Yaskawa INFORM job: OK_R2_O24B(90,0)KMOK.JBI

/JOB
//NAME OK_R2_O24B(90,0)KMOK
///FOLDERNAME X4
//POS
///NPOS 235,235,235,13,0,0
///TOOL 0
///POSTYPE PULSE
///PULSE
C00000=110421,-114568,-128442,17543,109310,-40994
C00001=110421,-114568,-128442,17543,109310,-40994
C00002=114535,-118016,-126260,17193,105500,-40103
C00003=116189,-118926,-125238,17079,104117,-39719
C00004=122470,-118801,-125267,16970,102934,-37675
C00005=122542,-119768,-123081,16831,101153,-37902
C00006=122470,-118801,-125267,16970,102934,-37675
C00007=116189,-118926,-125238,17079,104117,-39719
C00008=115768,-121709,-122546,16840,101244,-40278
C00009=119833,-121860,-122638,16796,100405,-38960
C00010=115768,-121709,-122546,16840,101244,-40278
C00011=116189,-118926,-125238,17079,104117,-39719
C00012=114535,-118016,-126260,17193,105500,-40103
C00013=110421,-114568,-128442,17543,109310,-40994
C00014=126378,-115954,-129597,-15290,109099,41008
C00015=122420,-119367,-127301,-14983,105339,40105
C00016=120830,-120251,-126232,-14883,103983,39719
C00017=114862,-120096,-125989,-14784,102865,37775
C00018=115075,-121077,-123808,-14669,101114,38064
C00019=114862,-120096,-125989,-14784,102865,37775
C00020=120830,-120251,-126232,-14883,103983,39719
C00021=121393,-120121,-122865,-14745,102140,40145
C00022=117360,-120220,-122765,-14697,101321,38836
C00023=121393,-120121,-122865,-14745,102140,40145
C00024=120830,-120251,-126232,-14883,103983,39719
C00025=122420,-119367,-127301,-14983,105339,40105
C00026=126378,-115954,-129597,-15290,109099,41008
C00027=68546,-106272,-120466,-15386,126682,61056
C00028=65872,-117617,-121364,-15125,121103,60799
C00029=65994,-124789,-121483,-14506,117628,61338
C00030=65994,-124776,-119887,-14364,116682,61464
C00031=64727,-121841,-121551,-15095,118908,60654
C00032=66354,-118147,-119193,-14717,119632,61205
C00033=63947,-125385,-121489,-15018,116968,60618
C00034=66354,-118147,-119193,-14717,119632,61205
C00035=67446,-114060,-119015,-14744,121753,61346
C00036=69995,-103128,-118158,-14981,127125,61604
C00037=43458,-109907,-123851,-22079,119459,51827
C00038=39582,-118676,-123782,-21672,114241,51374
C00039=37960,-121735,-123576,-21587,112243,51139
C00040=38039,-122241,-121246,-21299,110682,51473
C00041=37960,-121735,-123576,-21587,112243,51139
C00042=39439,-119560,-121458,-21353,112446,51673
C00043=35892,-124835,-123088,-21550,109947,50789
C00044=39439,-119560,-121458,-21353,112446,51673
C00045=41022,-116597,-121679,-21425,114395,51908
C00046=44803,-108153,-121807,-21787,119465,52368
C00047=46269,-104607,-116900,-14890,131588,81597
C00048=45575,-117487,-118566,-13929,126044,82146
C00049=45272,-122474,-119074,-13631,123805,82329
C00050=45097,-121786,-116375,-13476,122503,82429
C00051=45272,-122474,-119074,-13631,123805,82329
C00052=54794,-132635,-122270,-15461,117667,84057
C00053=51488,-139835,-124335,-16145,114686,83176
C00054=54794,-132635,-122270,-15461,117667,84057
C00055=54354,-108181,-111858,-18613,130239,82011
C00056=56948,-114588,-113873,-16794,128830,83498
C00057=54354,-108181,-111858,-18613,130239,82011
C00058=54354,-108181,-111858,-18613,105079,82011
C00059=125473,-127815,-125744,20402,114696,-66128
C00060=144354,-128645,-122856,20089,112993,-66444
C00061=144356,-128558,-121667,19978,112345,-66561
C00062=143692,-123642,-120175,20108,114021,-66516
C00063=144449,-128577,-122916,20120,113038,-66399
C00064=144368,-128510,-121483,19685,112887,-66475
C00065=144076,-129076,-121363,22700,108650,-60338
C00066=144065,-129172,-121967,22849,108765,-60054
C00067=145562,-127750,-121174,-10660,122518,-78224
C00068=145562,-127687,-120572,-10615,122186,-78189
C00069=144870,-122921,-119115,-11103,123620,-78631
C00070=145668,-127710,-121822,-10673,122944,-78224
C00071=145551,-127683,-120865,-10446,122273,-78190
C00072=145550,-127738,-121466,-10490,122609,-78224
C00073=145528,-127702,-122047,-10145,122795,-78223
C00074=145466,-127681,-122511,-8080,122804,-78067
C00075=145466,-127654,-121910,-8044,122451,-78039
C00076=144776,-122735,-120395,-8485,123961,-78447
C00077=145489,-127675,-123160,-8112,123205,-78089
C00078=145462,-127615,-121976,-8108,122518,-78051
C00079=145461,-127639,-122576,-8144,122872,-78079
C00080=145470,-127509,-122616,-9202,123100,-78187
C00081=145470,-127489,-122014,-9161,122745,-78155
C00082=144781,-122556,-120500,-9628,124248,-78581
C00083=145526,-127464,-123250,-9229,123515,-78201
C00084=145457,-127452,-122138,-8905,122802,-78142
C00085=145457,-127468,-122738,-8946,123159,-78173
C00086=145419,-127422,-123013,-7792,123191,-78085
C00087=145369,-127281,-122655,-6352,123642,-78005
C00088=145369,-127269,-122086,-6324,123301,-77983
C00089=144684,-122332,-120516,-6740,124807,-78367
C00090=145346,-127303,-123341,-6395,124049,-78040
C00091=145359,-127218,-122002,-6175,123337,-77977
C00092=145359,-127231,-122569,-6203,123677,-77998
C00093=145369,-127141,-122578,-7278,123283,-78064
C00094=145369,-127129,-121996,-7245,122933,-78039
C00095=144683,-122199,-120454,-7674,124442,-78435
C00096=145369,-127140,-123243,-7317,123689,-78093
C00097=145374,-127101,-121995,-7642,122781,-78062
C00098=145373,-127113,-122583,-7677,123134,-78088
C00099=145323,-127035,-122273,-5816,123755,-77984
C00100=145301,-126904,-121478,-4974,124764,-77984
C00101=145245,-126972,-122476,-3510,122733,-77759
C00102=145245,-126962,-121900,-3495,122385,-77747
C00103=144566,-122041,-120337,-3835,123918,-78081
C00104=145130,-127078,-123177,-3572,123105,-77819
C00105=145235,-126936,-121864,-3341,122099,-77723
C00106=145235,-126947,-122445,-3356,122451,-77734
C00107=145235,-126704,-121159,-4007,122972,-77833
C00108=145235,-126667,-120590,-3990,122642,-77820
C00109=144560,-121896,-119039,-4346,124100,-78159
C00110=145144,-126819,-121880,-4063,123351,-77885
C00111=145222,-126734,-121009,-3552,122070,-77754
C00112=143543,-128240,-121764,-3717,120897,-78337
C00113=144110,-127812,-122791,-3542,121772,-78139
C00114=145205,-126597,-125313,-3216,123991,-77765
C00115=78497,-119087,-126940,8466,133839,-13526
C00116=78488,-120793,-123596,8031,130934,-13800
C00117=78485,-121192,-122172,7887,129863,-13894
C00118=78455,-120845,-123307,7986,130735,-13833
C00119=77443,-125885,-123641,7190,128464,-14473
C00120=78479,-121212,-122221,7886,129884,-13896
C00121=78482,-120810,-123644,8031,130956,-13801
C00122=78491,-119095,-126985,8467,133863,-13526
C00123=78416,-117369,-129459,-12992,98157,-11559
C00124=78415,-119818,-126610,-12888,95218,-11250
C00125=78415,-120492,-125378,-12858,94139,-11138
C00126=77369,-125600,-126977,-12690,92378,-11308
C00127=78323,-119762,-126393,-12873,95102,-11269
C00128=78420,-120510,-125276,-12857,94070,-11129
C00129=78420,-119847,-126511,-12886,95145,-11241
C00130=78422,-117430,-129370,-12989,98073,-11548
C00131=84214,-85469,-118328,-4842,91147,-7442
C00132=74059,-12147,-76922,-1404,102997,-10572
C00133=133925,-71820,-61688,34619,64887,-29675
C00134=146663,-27707,-36323,28508,66625,-23960
C00135=151246,10085,-12654,25869,69264,-21358
C00136=159319,6651,-31532,14872,93153,-16403
C00137=161049,12617,-24359,-3467,88226,-17180
C00138=159447,19004,-16554,-3012,86648,-17647
C00139=159447,18503,-15222,-3010,85575,-17623
C00140=159447,19004,-16554,-3012,86648,-17647
C00141=159431,21694,-14016,-3008,86468,-17647
C00142=159447,19004,-16554,-3012,86648,-17647
C00143=160658,9490,-26043,14512,91068,-16216
C00144=162575,15072,-19202,14033,89453,-15776
C00145=163627,18223,-16292,13777,89114,-15470
C00146=163448,17947,-16551,13818,89157,-15522
C00147=163448,17469,-15177,13812,88099,-15642
C00148=162575,15072,-19202,14033,89453,-15776
C00149=162575,15072,-19202,14033,89453,-15776
C00150=161695,11045,-24734,14261,90891,-15899
C00151=160389,8166,-30281,14612,92983,-16078
C00152=166173,5650,-32242,20871,98882,-24992
C00153=168031,7092,-27994,20429,96691,-24741
C00154=171973,10796,-22826,19648,94585,-23756
C00155=171973,10387,-21674,19614,93717,-23897
C00156=171973,10796,-22826,19648,94585,-23756
C00157=173021,12834,-20995,19450,94274,-23449
C00158=171973,10796,-22826,19648,94585,-23756
C00159=169411,6672,-28771,20198,96619,-24285
C00160=169457,3960,-30994,23440,104028,-32838
C00161=170821,3186,-27404,27142,100799,-32384
C00162=170821,2940,-26605,27078,100248,-32515
C00163=170821,3186,-27404,27142,100799,-32384
C00164=171855,3656,-27002,27037,100474,-32081
C00165=170821,3186,-27404,27142,100799,-32384
C00166=171453,4765,-27678,27184,101480,-31989
C00167=155920,16768,-644,63423,123153,25810
C00168=153914,19171,3953,62063,123660,24610
C00169=157147,16214,3501,61820,121007,24650
C00170=157145,16372,4776,61403,120658,24311
C00171=157147,16214,3501,61820,121007,24650
C00172=158673,15787,3108,62073,120051,24962
C00173=157147,16214,3501,61820,121007,24650
C00174=154267,18481,3545,62056,123385,24630
C00175=160586,-4724,-32336,44114,114513,18408
C00176=159707,-1654,-23897,45976,117158,-10277
C00177=160426,-1772,-22346,45643,116076,-10462
C00178=160426,-1854,-21195,45350,115539,-10739
C00179=160426,-1772,-22346,45643,116076,-10462
C00180=161004,-2697,-23104,45705,115781,-10311
C00181=160426,-1772,-22346,45643,116076,-10462
C00182=174615,37008,-2722,25510,99744,-54261
C00183=172498,42405,8067,32730,102732,-53174
C00184=172498,42136,9154,32614,102046,-53379
C00185=172498,42405,8067,32730,102732,-53174
C00186=173166,39976,5518,32734,102755,-52903
C00187=172498,42405,8067,32730,102732,-53174
C00188=171464,48985,12939,32850,103438,-53371
C00189=169687,51444,12946,33160,105162,-53551
C00190=164203,-2216,-38598,32315,111910,-16095
C00191=166391,-1836,-35337,31828,109592,-15933
C00192=166612,13037,-20307,31307,106989,-15305
C00193=163905,10722,-24642,31867,110359,-16693
C00194=163023,10318,-23737,31712,110017,-17150
C00195=166579,13090,-20261,31308,106999,-15315
C00196=166501,27487,-9192,25512,104586,-16954
C00197=162952,34148,-2586,21763,97726,-15315
C00198=160142,17407,-18468,27124,95473,-4322
C00199=163018,-2778,-39064,26713,96671,-3025
C00200=164611,45054,6259,27542,116257,-62631
C00201=165962,40795,4672,27363,114755,-62481
C00202=169650,39468,5367,27407,112609,-61559
C00203=167727,42077,8101,27182,112908,-62250
C00204=168804,38233,1799,27701,114270,-61464
C00205=172646,46850,13078,27417,110817,-60826
C00206=175258,53962,20871,27351,108970,-60262
C00207=175286,54040,20958,27350,108949,-60256
C00208=176029,42421,9462,27228,100378,-50913
C00209=177057,44715,12834,27836,95407,-46661
C00210=174286,53569,18433,27340,100959,-51234
C00211=172614,55478,17651,27620,102791,-51416
C00212=158797,4213,-33188,27539,97918,-4223
C00213=160288,6924,-27895,27122,95799,-4194
C00214=161417,15198,-18304,26815,93980,-4213
C00215=160867,8461,-26639,27014,95638,-4024
C00216=160120,6892,-26748,27110,95204,-4392
C00217=161403,15259,-18249,26817,93982,-4218
C00218=160305,12086,-21204,20161,86451,4179
C00219=159689,11147,-21822,11042,81082,13112
C00220=158372,16674,-18680,7008,84648,12184
C00221=156002,16176,-19181,4250,84243,10833
C00222=159539,6079,-28636,11078,82663,13207
C00223=159574,4391,-38688,11011,87883,13681
C00224=158609,-20032,-50850,30856,115372,-43029
C00225=166404,-23641,-48444,30293,109810,-41499
C00226=167846,-166,-34046,28078,125353,-30479
C00227=167052,574,-32162,27620,124908,-30970
C00228=166419,-23641,-48461,30296,109814,-41492
C00229=164454,-27920,-49253,33885,103588,-43249
C00230=166369,-22686,-46969,33128,99976,-43386
C00231=169987,-10838,-39904,28688,98031,-37107
C00232=168025,-24410,-44140,30807,78602,-40011
C00233=160117,-23281,-55166,26476,98061,-35003
C00234=156670,-29522,-57811,32418,104336,-21012
BC00000=365719,492449,1075139
BC00001=365719,363190,1075139
BC00002=365719,363190,1075139
BC00003=365719,363190,1075139
BC00004=365719,363190,1075139
BC00005=365719,363190,1075139
BC00006=365719,363190,1075139
BC00007=365719,363190,1075139
BC00008=365719,363190,1075139
BC00009=365719,363190,1075139
BC00010=365719,363190,1075139
BC00011=365719,363190,1075139
BC00012=365719,363190,1075139
BC00013=365719,363190,1075139
BC00014=303651,361671,1075139
BC00015=303651,361671,1075139
BC00016=303651,361671,1075139
BC00017=303651,361671,1075139
BC00018=303651,361671,1075139
BC00019=303651,361671,1075139
BC00020=303651,361671,1075139
BC00021=303651,361671,1075139
BC00022=303651,361671,1075139
BC00023=303651,361671,1075139
BC00024=303651,361671,1075139
BC00025=303651,361671,1075139
BC00026=303651,361671,1075139
BC00027=337725,299685,1075139
BC00028=337725,299685,1075139
BC00029=337725,299685,1075139
BC00030=337725,299685,1075139
BC00031=337725,299685,1075139
BC00032=337725,299685,1075139
BC00033=337725,299685,1075139
BC00034=337725,299685,1075139
BC00035=337725,299685,1075139
BC00036=337725,299685,1075139
BC00037=224410,277346,1075139
BC00038=224410,277346,1075139
BC00039=224410,277346,1075139
BC00040=224410,277346,1075139
BC00041=224410,277346,1075139
BC00042=224410,277346,1075139
BC00043=224410,277346,1075139
BC00044=224410,277346,1075139
BC00045=224410,277346,1075139
BC00046=224410,277346,1075139
BC00047=171285,286904,1075139
BC00048=171285,286904,1075139
BC00049=171285,286904,1075139
BC00050=171285,286904,1075139
BC00051=171285,286904,1075139
BC00052=171285,286904,1075139
BC00053=171285,286904,1075139
BC00054=171285,286904,1075139
BC00055=171285,286904,1075139
BC00056=171285,286904,1075139
BC00057=171285,286904,1075139
BC00058=171285,286904,1075139
BC00059=269590,309617,1075139
BC00060=267805,314819,1075139
BC00061=267092,316899,1075139
BC00062=267092,316899,1075139
BC00063=267092,316899,1075139
BC00064=264540,316051,1075139
BC00065=269908,321406,1075139
BC00066=270630,320628,1075139
BC00067=229341,315661,1075139
BC00068=229396,316752,1075139
BC00069=229396,316752,1075139
BC00070=229396,316752,1075139
BC00071=236075,316791,1075139
BC00072=236027,315702,1075139
BC00073=249293,315797,1075139
BC00074=258915,315256,1075139
BC00075=258916,316331,1075139
BC00076=258916,316331,1075139
BC00077=258916,316331,1075139
BC00078=265201,316325,1075139
BC00079=265198,315250,1075139
BC00080=282635,315456,1075139
BC00081=282673,316525,1075139
BC00082=282673,316525,1075139
BC00083=282673,316525,1075139
BC00084=289448,316439,1075139
BC00085=289419,315369,1075139
BC00086=298136,315044,1075139
BC00087=312054,313301,1075139
BC00088=312047,314425,1075139
BC00089=312047,314425,1075139
BC00090=312047,314425,1075139
BC00091=318602,314234,1075139
BC00092=318613,313105,1075139
BC00093=336310,314307,1075139
BC00094=336328,315407,1075139
BC00095=336328,315407,1075139
BC00096=336328,315407,1075139
BC00097=342205,315848,1075139
BC00098=342175,314758,1075139
BC00099=344940,312597,1075139
BC00100=345730,309912,1075139
BC00101=367542,313335,1075139
BC00102=367491,314445,1075139
BC00103=367491,314445,1075139
BC00104=367491,314445,1075139
BC00105=374233,314799,1075139
BC00106=374293,313698,1075139
BC00107=391653,312000,1075139
BC00108=391630,313137,1075139
BC00109=391630,313137,1075139
BC00110=391630,313137,1075139
BC00111=394304,314202,1075139
BC00112=398158,315264,1075139
BC00113=398158,313163,1075139
BC00114=397780,307912,1075139
BC00115=322189,319410,1075139
BC00116=319334,319411,1075139
BC00117=318192,319412,1075139
BC00118=318192,319412,1075139
BC00119=318192,319412,1075139
BC00120=313651,319426,1075139
BC00121=314793,319425,1075139
BC00122=317648,319424,1075139
BC00123=260501,369489,1075139
BC00124=262854,366425,1075139
BC00125=263796,365199,1075139
BC00126=263796,365199,1075139
BC00127=263796,365199,1075139
BC00128=267671,365187,1075139
BC00129=266729,366413,1075139
BC00130=264376,369477,1075139
BC00131=264376,420432,1075139
BC00132=221796,515972,1075139
BC00133=202683,509615,271551
BC00134=202683,475987,185561
BC00135=202683,457833,139139
BC00136=138971,364074,115966
BC00137=138971,364074,115966
BC00138=138971,364074,115966
BC00139=138971,364074,115966
BC00140=138971,364074,115966
BC00141=138971,364074,115966
BC00142=138971,364074,115966
BC00143=138971,364074,115966
BC00144=138971,364074,115966
BC00145=138971,364074,115966
BC00146=138971,364074,115966
BC00147=138971,364074,115966
BC00148=138971,364074,115966
BC00149=138971,364074,115966
BC00150=138971,364074,115966
BC00151=138971,364074,115966
BC00152=150418,367609,116980
BC00153=150418,367609,116980
BC00154=150418,367608,116974
BC00155=150418,367608,116974
BC00156=150418,367608,116974
BC00157=150418,367608,116974
BC00158=150418,367608,116974
BC00159=150418,367609,116980
BC00160=147886,366442,115691
BC00161=147886,366442,115691
BC00162=147886,366442,115691
BC00163=147886,366442,115691
BC00164=147886,366442,115691
BC00165=147886,366442,115691
BC00166=163814,366442,115691
BC00167=140803,365672,114840
BC00168=140803,365672,114840
BC00169=140803,365673,114838
BC00170=140803,365673,114838
BC00171=140803,365673,114838
BC00172=140803,365673,114838
BC00173=140803,365673,114838
BC00174=140803,365672,114840
BC00175=149676,372426,112080
BC00176=161597,381499,108373
BC00177=161597,381499,108373
BC00178=161597,381499,108373
BC00179=161597,381499,108373
BC00180=161597,381499,108373
BC00181=161597,381499,108373
BC00182=245846,421854,91883
BC00183=245846,421854,91881
BC00184=245846,421854,91881
BC00185=245846,421854,91881
BC00186=245846,421854,91881
BC00187=245846,421854,91881
BC00188=245846,421854,91883
BC00189=245846,421854,91883
BC00190=140778,359593,95378
BC00191=140778,359593,95378
BC00192=140779,374954,95371
BC00193=140778,374954,95378
BC00194=140778,374954,95378
BC00195=140779,374954,95371
BC00196=140779,374954,95375
BC00197=140779,374954,95372
BC00198=140778,374954,95378
BC00199=140778,365135,95378
BC00200=224235,422354,101557
BC00201=224235,422354,101557
BC00202=224235,422354,101557
BC00203=224235,422354,101557
BC00204=224235,422354,101557
BC00205=224235,422354,101557
BC00206=224235,422354,101557
BC00207=224235,422354,101557
BC00208=224235,422354,101557
BC00209=224235,422354,101557
BC00210=224235,422354,101557
BC00211=224235,422354,101557
BC00212=135486,365173,95416
BC00213=135486,365173,95416
BC00214=135486,365173,95416
BC00215=135486,365173,95416
BC00216=135486,365173,95416
BC00217=135486,365173,95416
BC00218=135486,365173,95416
BC00219=135487,365173,95415
BC00220=135487,365173,95415
BC00221=135487,365173,95415
BC00222=135486,365173,95416
BC00223=135486,365173,95416
BC00224=147706,371102,95331
BC00225=147706,371102,95331
BC00226=147707,371103,95336
BC00227=147707,371103,95336
BC00228=147706,371102,95331
BC00229=147706,371102,95331
BC00230=147706,371102,95331
BC00231=147706,371102,95331
BC00232=147706,371102,95331
BC00233=147706,371102,95331
BC00234=147707,371103,95336
EC00000=-798156,-183832
EC00001=-798156,-183832
EC00002=-798156,-183832
EC00003=-798156,-183832
EC00004=-798156,-183832
EC00005=-798156,-183832
EC00006=-798156,-183832
EC00007=-798156,-183832
EC00008=-798156,-183832
EC00009=-798156,-183832
EC00010=-798156,-183832
EC00011=-798156,-183832
EC00012=-798156,-183832
EC00013=-798156,-183832
EC00014=-798156,-183832
EC00015=-798156,-183832
EC00016=-798156,-183832
EC00017=-798156,-183832
EC00018=-798156,-183832
EC00019=-798156,-183832
EC00020=-798156,-183832
EC00021=-798156,-183832
EC00022=-798156,-183832
EC00023=-798156,-183832
EC00024=-798156,-183832
EC00025=-798156,-183832
EC00026=-798156,-183832
EC00027=-798156,-183832
EC00028=-798156,-183832
EC00029=-798156,-183832
EC00030=-798156,-183832
EC00031=-798156,-183832
EC00032=-798156,-183832
EC00033=-798156,-183832
EC00034=-798156,-183832
EC00035=-798156,-183832
EC00036=-798156,-183832
EC00037=-798156,-183832
EC00038=-798156,-183832
EC00039=-798156,-183832
EC00040=-798156,-183832
EC00041=-798156,-183832
EC00042=-798156,-183832
EC00043=-798156,-183832
EC00044=-798156,-183832
EC00045=-798156,-183832
EC00046=-798156,-183832
EC00047=-798156,-183832
EC00048=-798156,-183832
EC00049=-798156,-183832
EC00050=-798156,-183832
EC00051=-798156,-183832
EC00052=-798156,-183832
EC00053=-798156,-183832
EC00054=-798156,-183832
EC00055=-798156,-183832
EC00056=-798156,-183832
EC00057=-798156,-183832
EC00058=-798156,-183832
EC00059=-798156,-183832
EC00060=-798156,-183832
EC00061=-798156,-183832
EC00062=-798156,-183832
EC00063=-798156,-183832
EC00064=-798156,-183832
EC00065=-798156,-183832
EC00066=-798156,-183832
EC00067=-798156,-183832
EC00068=-798156,-183832
EC00069=-798156,-183832
EC00070=-798156,-183832
EC00071=-798156,-183832
EC00072=-798156,-183832
EC00073=-798156,-183832
EC00074=-798156,-183832
EC00075=-798156,-183832
EC00076=-798156,-183832
EC00077=-798156,-183832
EC00078=-798156,-183832
EC00079=-798156,-183832
EC00080=-798156,-183832
EC00081=-798156,-183832
EC00082=-798156,-183832
EC00083=-798156,-183832
EC00084=-798156,-183832
EC00085=-798156,-183832
EC00086=-798156,-183832
EC00087=-798156,-183832
EC00088=-798156,-183832
EC00089=-798156,-183832
EC00090=-798156,-183832
EC00091=-798156,-183832
EC00092=-798156,-183832
EC00093=-798156,-183832
EC00094=-798156,-183832
EC00095=-798156,-183832
EC00096=-798156,-183832
EC00097=-798156,-183832
EC00098=-798156,-183832
EC00099=-798156,-183832
EC00100=-798156,-183832
EC00101=-798156,-183832
EC00102=-798156,-183832
EC00103=-798156,-183832
EC00104=-798156,-183832
EC00105=-798156,-183832
EC00106=-798156,-183832
EC00107=-798156,-183832
EC00108=-798156,-183832
EC00109=-798156,-183832
EC00110=-798156,-183832
EC00111=-798156,-183832
EC00112=-798156,-183832
EC00113=-798156,-183832
EC00114=-798156,-183832
EC00115=-798156,-183832
EC00116=-798156,-183832
EC00117=-798156,-183832
EC00118=-798156,-183832
EC00119=-798156,-183832
EC00120=-798156,-183832
EC00121=-798156,-183832
EC00122=-798156,-183832
EC00123=-798156,-183832
EC00124=-798156,-183832
EC00125=-798156,-183832
EC00126=-798156,-183832
EC00127=-798156,-183832
EC00128=-798156,-183832
EC00129=-798156,-183832
EC00130=-798156,-183832
EC00131=-798156,-183832
EC00132=-798156,-183832
EC00133=-798156,-183832
EC00134=-798156,-183832
EC00135=-798156,-183832
EC00136=-798156,-183832
EC00137=-798156,-183832
EC00138=-798156,-183832
EC00139=-798156,-183832
EC00140=-798156,-183832
EC00141=-798156,-183832
EC00142=-798156,-183832
EC00143=-798156,-183832
EC00144=-798156,-183832
EC00145=-798156,-183832
EC00146=-798156,-183832
EC00147=-798156,-183832
EC00148=-798156,-183832
EC00149=-798156,-183832
EC00150=-798156,-183832
EC00151=-798156,-183832
EC00152=-798156,-183832
EC00153=-798156,-183832
EC00154=-798154,-183833
EC00155=-798154,-183833
EC00156=-798154,-183833
EC00157=-798154,-183833
EC00158=-798154,-183833
EC00159=-798156,-183832
EC00160=-798156,-183832
EC00161=-798156,-183832
EC00162=-798156,-183832
EC00163=-798156,-183832
EC00164=-798156,-183832
EC00165=-798156,-183832
EC00166=-798156,-183832
EC00167=-798156,-183832
EC00168=-798156,-183832
EC00169=-798154,-183832
EC00170=-798154,-183832
EC00171=-798154,-183832
EC00172=-798154,-183832
EC00173=-798154,-183832
EC00174=-798156,-183832
EC00175=-798156,-183832
EC00176=-798156,-183832
EC00177=-798156,-183832
EC00178=-798156,-183832
EC00179=-798156,-183832
EC00180=-798156,-183832
EC00181=-798156,-183832
EC00182=-798156,-183832
EC00183=-798154,-183833
EC00184=-798154,-183833
EC00185=-798154,-183833
EC00186=-798154,-183833
EC00187=-798154,-183833
EC00188=-798156,-183832
EC00189=-798156,-183832
EC00190=-798156,-183832
EC00191=-798156,-183832
EC00192=-798154,-183833
EC00193=-798156,-183832
EC00194=-798156,-183832
EC00195=-798154,-183833
EC00196=-798155,-183833
EC00197=-798154,-183834
EC00198=-798156,-183832
EC00199=-798156,-183832
EC00200=-798156,-183832
EC00201=-798156,-183832
EC00202=-798156,-183832
EC00203=-798156,-183832
EC00204=-798156,-183832
EC00205=-798156,-183832
EC00206=-798156,-183832
EC00207=-798156,-183832
EC00208=-798156,-183832
EC00209=-798156,-183832
EC00210=-798156,-183832
EC00211=-798156,-183832
EC00212=-798156,-183832
EC00213=-798156,-183832
EC00214=-798156,-183832
EC00215=-798156,-183832
EC00216=-798156,-183832
EC00217=-798156,-183832
EC00218=-798156,-183832
EC00219=-798155,-183833
EC00220=-798155,-183833
EC00221=-798155,-183833
EC00222=-798156,-183832
EC00223=-798156,-183832
EC00224=-798153,-183833
EC00225=-798153,-183833
EC00226=-798156,-183832
EC00227=-798156,-183832
EC00228=-798153,-183833
EC00229=-798153,-183833
EC00230=-798153,-183833
EC00231=-798153,-183833
EC00232=-798153,-183833
EC00233=-798153,-183833
EC00234=-798156,-183832
///POSTYPE BASE
///RECTAN
///RCONF 0,0,0,0,1,0,0,0,0,0,0,0,0,0,0,0,0,0,0,0,0,0,0,0
P00006=2.006,1.622,-0.565,0.0000,0.0000,0.0000
P00021=0.073,2.058,-0.109,0.0000,0.0000,0.0000
P00022=2.006,1.622,-0.565,0.0000,0.0000,0.0000
///RCONF 0,0,0,0,0,0,0,0,0,0,0,0,0,0,0,0,0,0,0,0,0,0,0,0
P00023=-2.957,-4.083,2.762,0.0000,0.0000,0.0000
P00024=-1.466,-0.226,-0.419,0.0000,0.0000,0.0000
P00025=3.643,0.007,-2.585,0.0000,0.0000,0.0000
P00026=2.644,0.055,-2.583,0.0000,0.0000,0.0000
P00027=2.278,0.099,-4.210,0.0000,0.0000,0.0000
P00031=-0.170,0.039,-0.647,0.0000,0.0000,0.0000
P00032=-0.423,0.157,3.222,0.0000,0.0000,0.0000
P00033=0.854,-1.099,3.047,0.0000,0.0000,0.0000
///RCONF 0,0,0,0,1,0,0,0,0,0,0,0,0,0,0,0,0,0,0,0,0,0,0,0
P00034=-8.151,9.743,-4.393,0.0000,0.0000,0.0000
///RCONF 0,0,0,0,0,0,0,0,0,0,0,0,0,0,0,0,0,0,0,0,0,0,0,0
P00035=0.390,-0.027,1.040,0.0000,0.0000,0.0000
//INST
///DATE 2024/11/18 12:50
///ATTR SC,RW
///GROUP1 RB1,BS1
///GROUP2 ST1
NOP
'OK_r2_O24B(90,0)
'
'brak tej czesci na razie
'Path S3723
SFTOF3D
MOVJ C00000 BC00000 VJ=100.00  +MOVJ EC00000 VJ=100.00
JUMP *LABEL
MOVJ C00001 BC00001 VJ=100.00  +MOVJ EC00001 VJ=100.00
MOVL C00002 BC00002 V=400.0  +MOVJ EC00002 VJ=100.00
SMOVL C00003 BC00003 V=100.0  +MOVJ EC00003
'BRAK DETALU
PAUSE
SMOVL C00004 BC00004 V=60.0  +MOVJ EC00004
SREFP 3 C00005 BC00005  +REFP EC00005
CALL JOB:SEARCH-R1-S13D
SET P031 P006
SFTON3D P031
SMOVL C00006 BC00006 V=60.0  +MOVJ EC00006
SMOVL C00007 BC00007 V=100.0  +MOVJ EC00007
SMOVL C00008 BC00008 V=60.0  +MOVJ EC00008
SREFP 3 C00009 BC00009  +REFP EC00009
CALL JOB:SEARCH-R1-S13D
SET P031 P006
SFTON3D P031
SMOVL C00010 BC00010 V=60.0  +MOVJ EC00010
SMOVL C00011 BC00011 V=100.0  +MOVJ EC00011
MOVL C00012 BC00012 V=400.0  +MOVJ EC00012 VJ=100.00
MOVL C00013 BC00013 V=1000.0  +MOVJ EC00013 VJ=100.00
'Path S3724
SFTOF3D
MOVJ C00014 BC00014 VJ=100.00  +MOVJ EC00014 VJ=100.00
MOVL C00015 BC00015 V=400.0  +MOVJ EC00015 VJ=100.00
SMOVL C00016 BC00016 V=100.0  +MOVJ EC00016
SMOVL C00017 BC00017 V=60.0  +MOVJ EC00017
SREFP 3 C00018 BC00018  +REFP EC00018
CALL JOB:SEARCH-R1-S13D
SET P032 P006
SFTON3D P032
SMOVL C00019 BC00019 V=60.0  +MOVJ EC00019
SMOVL C00020 BC00020 V=100.0  +MOVJ EC00020
SMOVL C00021 BC00021 V=60.0  +MOVJ EC00021
SREFP 3 C00022 BC00022  +REFP EC00022
CALL JOB:SEARCH-R1-S13D
SET P032 P006
SFTON3D P032
SMOVL C00023 BC00023 V=60.0  +MOVJ EC00023
SMOVL C00024 BC00024 V=100.0  +MOVJ EC00024
MOVL C00025 BC00025 V=400.0  +MOVJ EC00025 VJ=100.00
MOVL C00026 BC00026 V=1000.0  +MOVJ EC00026 VJ=100.00
'Path S3725
SFTOF3D
MOVJ C00027 BC00027 VJ=100.00  +MOVJ EC00027 VJ=100.00
MOVL C00028 BC00028 V=400.0  +MOVJ EC00028 VJ=100.00
SMOVL C00029 BC00029 V=60.0  +MOVJ EC00029
SREFP 3 C00030 BC00030  +REFP EC00030
CALL JOB:SEARCH-R1-S13D
SET P034 P006
SFTON3D P034
SMOVL C00031 BC00031 V=60.0  +MOVJ EC00031
SMOVL C00032 BC00032 V=60.0  +MOVJ EC00032
SREFP 3 C00033 BC00033  +REFP EC00033
CALL JOB:SEARCH-R1-S13D
SET P034 P006
SFTON3D P034
SMOVL C00034 BC00034 V=60.0  +MOVJ EC00034
MOVL C00035 BC00035 V=400.0  +MOVJ EC00035 VJ=100.00
MOVL C00036 BC00036 V=1000.0  +MOVJ EC00036 VJ=100.00
'Path S3726
SFTOF3D
MOVJ C00037 BC00037 VJ=100.00  +MOVJ EC00037 VJ=100.00
MOVL C00038 BC00038 V=400.0  +MOVJ EC00038 VJ=100.00
SMOVL C00039 BC00039 V=60.0  +MOVJ EC00039
SREFP 3 C00040 BC00040  +REFP EC00040
CALL JOB:SEARCH-R1-S13D
SET P035 P006
SFTON3D P035
SMOVL C00041 BC00041 V=60.0  +MOVJ EC00041
SMOVL C00042 BC00042 V=60.0  +MOVJ EC00042
SREFP 3 C00043 BC00043  +REFP EC00043
CALL JOB:SEARCH-R1-S13D
SET P035 P006
SFTON3D P035
SMOVL C00044 BC00044 V=60.0  +MOVJ EC00044
MOVL C00045 BC00045 V=400.0  +MOVJ EC00045 VJ=100.00
MOVL C00046 BC00046 V=1000.0  +MOVJ EC00046 VJ=100.00
'Path S3727
SFTOF3D
MOVJ C00047 BC00047 VJ=100.00  +MOVJ EC00047 VJ=100.00
MOVL C00048 BC00048 V=400.0  +MOVJ EC00048 VJ=100.00
SMOVL C00049 BC00049 V=60.0  +MOVJ EC00049
SREFP 3 C00050 BC00050  +REFP EC00050
CALL JOB:SEARCH-R1-S13D
SET P033 P006
SFTON3D P033
SMOVL C00051 BC00051 V=60.0  +MOVJ EC00051
SMOVL C00052 BC00052 V=60.0  +MOVJ EC00052
SREFP 3 C00053 BC00053  +REFP EC00053
CALL JOB:SEARCH-R1-S13D
SET P033 P006
SFTON3D P033
SMOVL C00054 BC00054 V=60.0  +MOVJ EC00054
SMOVL C00055 BC00055 V=60.0  +MOVJ EC00055
SREFP 3 C00056 BC00056  +REFP EC00056
CALL JOB:SEARCH-R1-S13D
SET P033 P006
SFTON3D P033
MOVJ C00057 BC00057 VJ=50.00  +MOVJ EC00057 VJ=50.00
MOVJ C00058 BC00058 VJ=50.00  +MOVJ EC00058 VJ=50.00
'Path W3728
SFTOF3D
SFTON3D P033
MOVJ C00059 BC00059 VJ=100.00  +MOVJ EC00059 VJ=100.00
SMOVL C00060 BC00060 V=400.0  +MOVJ EC00060
SMOVL C00061 BC00061 V=100.0 PL=0  +MOVJ EC00061
SREFP 1 C00062 BC00062  +REFP EC00062
SREFP 2 C00063 BC00063  +REFP EC00063
MACRO1 MJ#(0) ARGF0
ARCON
SMOVL C00064 BC00064 V=10.0  +MOVJ EC00064
SMOVL C00065 BC00065 V=10.0  +MOVJ EC00065
ARCOF
SMOVL C00066 BC00066 V=100.0  +MOVJ EC00066
SMOVL C00067 BC00067 V=100.0  +MOVJ EC00067
SMOVL C00068 BC00068 V=100.0 PL=0  +MOVJ EC00068
SREFP 1 C00069 BC00069  +REFP EC00069
SREFP 2 C00070 BC00070  +REFP EC00070
MACRO1 MJ#(0) ARGF0
ARCON
SMOVL C00071 BC00071 V=10.0  +MOVJ EC00071
ARCOF
SMOVL C00072 BC00072 V=100.0  +MOVJ EC00072
SFTON3D P035
SMOVL C00073 BC00073 V=100.0  +MOVJ EC00073
SMOVL C00074 BC00074 V=100.0  +MOVJ EC00074
SMOVL C00075 BC00075 V=100.0 PL=0  +MOVJ EC00075
SREFP 1 C00076 BC00076  +REFP EC00076
SREFP 2 C00077 BC00077  +REFP EC00077
MACRO1 MJ#(0) ARGF0
ARCON
SMOVL C00078 BC00078 V=10.0  +MOVJ EC00078
ARCOF
SMOVL C00079 BC00079 V=100.0  +MOVJ EC00079
SMOVL C00080 BC00080 V=100.0  +MOVJ EC00080
SMOVL C00081 BC00081 V=100.0 PL=0  +MOVJ EC00081
SREFP 1 C00082 BC00082  +REFP EC00082
SREFP 2 C00083 BC00083  +REFP EC00083
MACRO1 MJ#(0) ARGF0
ARCON
SMOVL C00084 BC00084 V=10.0  +MOVJ EC00084
ARCOF
SMOVL C00085 BC00085 V=100.0  +MOVJ EC00085
SMOVL C00086 BC00086 V=100.0  +MOVJ EC00086
SMOVL C00087 BC00087 V=100.0  +MOVJ EC00087
SMOVL C00088 BC00088 V=100.0 PL=0  +MOVJ EC00088
SREFP 1 C00089 BC00089  +REFP EC00089
SREFP 2 C00090 BC00090  +REFP EC00090
MACRO1 MJ#(0) ARGF0
ARCON
SMOVL C00091 BC00091 V=10.0  +MOVJ EC00091
ARCOF
SMOVL C00092 BC00092 V=100.0  +MOVJ EC00092
SMOVL C00093 BC00093 V=100.0  +MOVJ EC00093
SMOVL C00094 BC00094 V=100.0 PL=0  +MOVJ EC00094
SREFP 1 C00095 BC00095  +REFP EC00095
SREFP 2 C00096 BC00096  +REFP EC00096
MACRO1 MJ#(0) ARGF0
ARCON
SMOVL C00097 BC00097 V=10.0  +MOVJ EC00097
ARCOF
SMOVL C00098 BC00098 V=100.0  +MOVJ EC00098
SMOVL C00099 BC00099 V=100.0  +MOVJ EC00099
SMOVL C00100 BC00100 V=100.0  +MOVJ EC00100
SFTON3D P034
SMOVL C00101 BC00101 V=100.0  +MOVJ EC00101
SMOVL C00102 BC00102 V=100.0 PL=0  +MOVJ EC00102
SREFP 1 C00103 BC00103  +REFP EC00103
SREFP 2 C00104 BC00104  +REFP EC00104
MACRO1 MJ#(0) ARGF0
ARCON
SMOVL C00105 BC00105 V=10.0  +MOVJ EC00105
ARCOF
SMOVL C00106 BC00106 V=100.0  +MOVJ EC00106
SMOVL C00107 BC00107 V=100.0  +MOVJ EC00107
SMOVL C00108 BC00108 V=100.0 PL=0  +MOVJ EC00108
SREFP 1 C00109 BC00109  +REFP EC00109
SREFP 2 C00110 BC00110  +REFP EC00110
MACRO1 MJ#(0) ARGF0
ARCON
SMOVL C00111 BC00111 V=10.0  +MOVJ EC00111
SMOVL C00112 BC00112 V=10.0  +MOVJ EC00112
ARCOF
SMOVL C00113 BC00113 V=400.0  +MOVJ EC00113
SMOVL C00114 BC00114 V=1000.0  +MOVJ EC00114
SFTOF3D
'Path W3729
SFTOF3D
SFTON3D P031
MOVJ C00115 BC00115 VJ=100.00  +MOVJ EC00115 VJ=100.00
SMOVL C00116 BC00116 V=400.0  +MOVJ EC00116
SMOVL C00117 BC00117 V=100.0 PL=0  +MOVJ EC00117
SREFP 1 C00118 BC00118  +REFP EC00118
SREFP 2 C00119 BC00119  +REFP EC00119
MACRO1 MJ#(0) ARGF0
ARCON
SMOVL C00120 BC00120 V=10.0  +MOVJ EC00120
ARCOF
SMOVL C00121 BC00121 V=400.0  +MOVJ EC00121
SMOVL C00122 BC00122 V=1000.0  +MOVJ EC00122
SFTOF3D
'Path W3730
SFTOF3D
SFTON3D P032
MOVJ C00123 BC00123 VJ=100.00  +MOVJ EC00123 VJ=100.00
SMOVL C00124 BC00124 V=400.0  +MOVJ EC00124
SMOVL C00125 BC00125 V=100.0 PL=0  +MOVJ EC00125
SREFP 1 C00126 BC00126  +REFP EC00126
SREFP 2 C00127 BC00127  +REFP EC00127
MACRO1 MJ#(0) ARGF0
ARCON
SMOVL C00128 BC00128 V=10.0  +MOVJ EC00128
ARCOF
SMOVL C00129 BC00129 V=400.0  +MOVJ EC00129
SMOVL C00130 BC00130 V=1000.0  +MOVJ EC00130
SFTOF3D
MOVJ C00131 BC00131 VJ=100.00  +MOVJ EC00131 VJ=100.00
MOVJ C00132 BC00132 VJ=100.00  +MOVJ EC00132 VJ=100.00
'dotad odkoment
'down
*LABEL
MOVJ C00133 BC00133 VJ=100.00  +MOVJ EC00133 VJ=100.00
MOVJ C00134 BC00134 VJ=100.00  +MOVJ EC00134 VJ=100.00
MOVJ C00135 BC00135 VJ=15.00  +MOVJ EC00135 VJ=100.00
'Path S3731
SFTOF3D
MOVJ C00136 BC00136 VJ=30.00  +MOVJ EC00136 VJ=100.00
MOVJ C00137 BC00137 VJ=30.00  +MOVJ EC00137 VJ=0.78
SMOVL C00138 BC00138 V=166.7  +MOVJ EC00138
SREFP 3 C00139 BC00139  +REFP EC00139
CALL JOB:SEARCH-R1-S13D
SET P025 P006
SFTON3D P025
SMOVL C00140 BC00140 V=100.0  +MOVJ EC00140
SREFP 3 C00141 BC00141  +REFP EC00141
CALL JOB:SEARCH-R1-S13D
SET P025 P006
SFTON3D P025
SMOVL C00142 BC00142 V=250.0  +MOVJ EC00142
SFTOF3D
MOVL C00143 BC00143 V=400.0  +MOVJ EC00143 VJ=100.00
SMOVL C00144 BC00144 V=100.0  +MOVJ EC00144
SREFP 3 C00145 BC00145  +REFP EC00145
CALL JOB:SEARCH-R1-S13D
SET P021 P006
SFTON3D P021
SMOVL C00146 BC00146 V=83.3  +MOVJ EC00146
SREFP 3 C00147 BC00147  +REFP EC00147
CALL JOB:SEARCH-R1-S13D
SET P021 P006
SFTON3D P021
SMOVL C00148 BC00148 V=100.0  +MOVJ EC00148
SMOVL C00149 BC00149 V=100.0  +MOVJ EC00149
MOVL C00150 BC00150 V=400.0  +MOVJ EC00150 VJ=100.00
MOVL C00151 BC00151 V=1000.0  +MOVJ EC00151 VJ=100.00
'Path S3732
SFTOF3D
MOVJ C00152 BC00152 VJ=100.00  +MOVJ EC00152 VJ=100.00
MOVL C00153 BC00153 V=400.0  +MOVJ EC00153 VJ=100.00
SMOVL C00154 BC00154 V=100.0  +MOVJ EC00154
SREFP 3 C00155 BC00155  +REFP EC00155
CALL JOB:SEARCH-R1-S13D
SET P022 P006
SFTON3D P022
SMOVL C00156 BC00156 V=100.0  +MOVJ EC00156
SREFP 3 C00157 BC00157  +REFP EC00157
CALL JOB:SEARCH-R1-S13D
SET P022 P006
SFTON3D P022
SMOVL C00158 BC00158 V=100.0  +MOVJ EC00158
SFTOF3D
MOVL C00159 BC00159 V=400.0  +MOVJ EC00159 VJ=100.00
MOVL C00160 BC00160 V=500.0  +MOVJ EC00160 VJ=100.00
SMOVL C00161 BC00161 V=166.7  +MOVJ EC00161
SREFP 3 C00162 BC00162  +REFP EC00162
CALL JOB:SEARCH-R1-S13D
SET P027 P006
SFTON3D P027
SMOVL C00163 BC00163 V=100.0  +MOVJ EC00163
SREFP 3 C00164 BC00164  +REFP EC00164
CALL JOB:SEARCH-R1-S13D
SET P027 P006
SFTON3D P027
SMOVL C00165 BC00165 V=166.7  +MOVJ EC00165
'Path S3733
SFTOF3D
MOVJ C00166 BC00166 VJ=15.00  +MOVJ EC00166 VJ=0.78
MOVJ C00167 BC00167 VJ=15.00  +MOVJ EC00167 VJ=15.00
MOVL C00168 BC00168 V=400.0  +MOVJ EC00168 VJ=100.00
SMOVL C00169 BC00169 V=166.7  +MOVJ EC00169
SREFP 3 C00170 BC00170  +REFP EC00170
CALL JOB:SEARCH-R1-S13D
SET P023 P006
SFTON3D P023
SMOVL C00171 BC00171 V=100.0  +MOVJ EC00171
SREFP 3 C00172 BC00172  +REFP EC00172
CALL JOB:SEARCH-R1-S13D
SET P023 P006
SFTON3D P023
SMOVL C00173 BC00173 V=166.7  +MOVJ EC00173
MOVL C00174 BC00174 V=400.0  +MOVJ EC00174 VJ=100.00
'Path S3734
SFTOF3D
MOVJ C00175 BC00175 VJ=15.00  +MOVJ EC00175 VJ=15.00
MOVJ C00176 BC00176 VJ=20.00  +MOVJ EC00176 VJ=0.78
SMOVL C00177 BC00177 V=166.7  +MOVJ EC00177
SREFP 3 C00178 BC00178  +REFP EC00178
CALL JOB:SEARCH-R1-S13D
SET P026 P006
SFTON3D P026
SMOVL C00179 BC00179 V=166.7  +MOVJ EC00179
SREFP 3 C00180 BC00180  +REFP EC00180
CALL JOB:SEARCH-R1-S13D
SET P026 P006
SFTON3D P026
SMOVL C00181 BC00181 V=166.7  +MOVJ EC00181
MOVL C00182 BC00182 V=400.0  +MOVJ EC00182 VJ=100.00
SMOVL C00183 BC00183 V=100.0  +MOVJ EC00183
SREFP 3 C00184 BC00184  +REFP EC00184
CALL JOB:SEARCH-R1-S13D
SET P024 P006
SFTON3D P024
SMOVL C00185 BC00185 V=100.0  +MOVJ EC00185
SREFP 3 C00186 BC00186  +REFP EC00186
CALL JOB:SEARCH-R1-S13D
SET P024 P006
SFTON3D P024
SMOVL C00187 BC00187 V=100.0  +MOVJ EC00187
MOVL C00188 BC00188 V=400.0  +MOVJ EC00188 VJ=100.00
MOVL C00189 BC00189 V=1000.0  +MOVJ EC00189 VJ=100.00
'Path W3735
SFTOF3D
MOVJ C00190 BC00190 VJ=100.00  +MOVJ EC00190 VJ=100.00
SMOVL C00191 BC00191 V=400.0  +MOVJ EC00191
SFTON3D P027
SMOVL C00192 BC00192 V=166.7 PL=0  +MOVJ EC00192
SREFP 1 C00193 BC00193  +REFP EC00193
SREFP 2 C00194 BC00194  +REFP EC00194
MACRO1 MJ#(0) ARGF21
ARCON
SWVON WEV#(100)
SMOVC C00195 BC00195 V=8.3  +MOVJ EC00195
SFTON3D P022
SMOVC C00196 BC00196 V=8.3  +MOVJ EC00196
SFTON3D P021
SMOVC C00197 BC00197 V=8.3  +MOVJ EC00197
ARCOF
SWVOF
SMOVL C00198 BC00198 V=400.0  +MOVJ EC00198
SMOVL C00199 BC00199 V=1000.0  +MOVJ EC00199
SFTOF3D
'Path W3737
SFTOF3D
SFTON3D P024
MOVJ C00200 BC00200 VJ=100.00  +MOVJ EC00200 VJ=100.00
SMOVL C00201 BC00201 V=400.0  +MOVJ EC00201
SMOVL C00202 BC00202 V=166.7 PL=0  +MOVJ EC00202
SREFP 1 C00203 BC00203  +REFP EC00203
SREFP 2 C00204 BC00204  +REFP EC00204
MACRO1 MJ#(0) ARGF21
ARCON
SWVON WEV#(100)
SMOVL C00205 BC00205 V=8.3  +MOVJ EC00205
SMOVL C00206 BC00206 V=8.3  +MOVJ EC00206
SMOVC C00207 BC00207 V=8.3  +MOVJ EC00207
SFTON3D P026
SMOVC C00208 BC00208 V=8.3  +MOVJ EC00208
SMOVC C00209 BC00209 V=8.3  +MOVJ EC00209
ARCOF
SWVOF
SMOVL C00210 BC00210 V=400.0  +MOVJ EC00210
SMOVL C00211 BC00211 V=1000.0  +MOVJ EC00211
SFTOF3D
'Path W3736
SFTOF3D
SFTON3D P021
MOVJ C00212 BC00212 VJ=100.00  +MOVJ EC00212 VJ=100.00
SMOVL C00213 BC00213 V=400.0  +MOVJ EC00213
SFTON3D P021
SMOVL C00214 BC00214 V=166.7 PL=0  +MOVJ EC00214
SREFP 1 C00215 BC00215  +REFP EC00215
SREFP 2 C00216 BC00216  +REFP EC00216
MACRO1 MJ#(0) ARGF21
ARCON
SWVON WEV#(100)
SMOVC C00217 BC00217 V=8.3  +MOVJ EC00217
SMOVC C00218 BC00218 V=8.3  +MOVJ EC00218
SFTON3D P025
SMOVC C00219 BC00219 V=8.3  +MOVJ EC00219
SMOVC C00220 BC00220 V=8.3  +MOVJ EC00220
SMOVL C00221 BC00221 V=8.3  +MOVJ EC00221
ARCOF
SWVOF
SFTOF3D
SMOVL C00222 BC00222 V=400.0  +MOVJ EC00222
SMOVL C00223 BC00223 V=1000.0  +MOVJ EC00223
SFTOF3D
'Path W3738
SFTOF3D
SFTON3D P026
SMOVL C00224 BC00224 V=583.3  +MOVJ EC00224
SMOVL C00225 BC00225 V=166.7 PL=0  +MOVJ EC00225
SREFP 1 C00226 BC00226  +REFP EC00226
SREFP 2 C00227 BC00227  +REFP EC00227
MACRO1 MJ#(0) ARGF21
ARCON
SWVON WEV#(100)
SMOVC C00228 BC00228 V=8.3  +MOVJ EC00228
SMOVC C00229 BC00229 V=8.3  +MOVJ EC00229
SFTON3D P023
SMOVC C00230 BC00230 V=8.3  +MOVJ EC00230
SFTON3D P027
SMOVC C00231 BC00231 V=8.3  +MOVJ EC00231
SMOVC C00232 BC00232 V=8.3  +MOVJ EC00232
ARCOF
SWVOF
SFTOF3D
SMOVL C00233 BC00233 V=400.0  +MOVJ EC00233
SMOVL C00234 BC00234 V=1000.0  +MOVJ EC00234
SFTOF3D
END
